TYPE MotorOutput :
STRUCT
	ConveyorForward : BOOL;
	ConveyorBackward : BOOL;
	ConveyorStop : BOOL;
	ConveyorSpeed : UDINT;
END_STRUCT
END_TYPE

(* stored: Version 1.1.0.1
   DUT MotorOutput: Id {f28daf18-d411-4e0a-9f93-013fe10c5e47} *)
